{attribute 'linkalways'} 
{attribute 'no_explicit_call' := 'This FB is a CLASS and must be accessed using methods or properties'}
{attribute 'enable_dynamic_creation'}
FUNCTION_BLOCK JsonDeserializer EXTENDS Disposable IMPLEMENTS I_JsonDeserializer
VAR
	jsonParser : JsonDomParser;
	root : SJsonValue;
	garbageCollector : DeserializerGarbageCollector;
	nullNode : JsonDeserializerNullNode(THIS^);
	rootNode : I_Deserializer := nullNode;
	eventEmitter : EventEmitter;
END_VAR

METHOD PUBLIC Clone : I_Deserializer
VAR
	pClone : POINTER TO JsonDeserializer;
	jsonSize : UDINT;
	pJsonString : POINTER TO STRING;
END_VAR
pClone := __NEW(JsonDeserializer);
Clone := pClone^;

jsonSize := jsonParser.GetDocumentLength();

IF jsonSize = 0 THEN
	// no further cloning to do. 
	RETURN;
END_IF

pJsonString := __NEW(BYTE, jsonSize);

IF jsonParser.CopyDocument(pJsonString^, jsonSize) = 0 THEN
	__DELETE(pJsonString);
	RETURN;
END_IF

pClone^.TryLoad(pJsonString^);
__DELETE(pJsonString);
END_METHOD

METHOD PROTECTED CreateDeserializer : I_Deserializer
VAR_INPUT
	DeserializerRoot : SJsonValue;
END_VAR
VAR 
	pNode : POINTER TO JsonDeserializerNode;
END_VAR
pNode := __NEW(JsonDeserializerNode(
	ParentJsonDeserializer := THIS^,
	ParentJsonDomParser := jsonParser, 
	NodeRoot := DeserializerRoot, 
	ParentGarbageCollector := garbageCollector, 
	ParentNullDeserializer := nullNode)
);

CreateDeserializer := pNode^;
END_METHOD

METHOD PRIVATE EmitChangedEvent
VAR
	pJsonDeserializerChangedEvent : POINTER TO JsonDeserializerChangedEvent;
END_VAR
pJsonDeserializerChangedEvent := __NEW(JsonDeserializerChangedEvent(Target := THIS^));
eventEmitter.Emit('OnChanged', pJsonDeserializerChangedEvent^);
pJsonDeserializerChangedEvent^.Dispose();
END_METHOD

METHOD PRIVATE EmitDisposedEvent
VAR
	pJsonDeserializerDisposedEvent : POINTER TO JsonDeserializerDisposedEvent;
END_VAR
pJsonDeserializerDisposedEvent := __NEW(JsonDeserializerDisposedEvent(Target := THIS^));
eventEmitter.Emit('OnDisposed', pJsonDeserializerDisposedEvent^);
pJsonDeserializerDisposedEvent^.Dispose();
END_METHOD

METHOD FB_exit : BOOL
VAR_INPUT
	bInCopyCode : BOOL; // if TRUE, the exit method is called for exiting an instance that is copied afterwards (online change).
END_VAR
IF bInCopyCode THEN
	RETURN;
END_IF

Reset();
EmitDisposedEvent();
END_METHOD

METHOD GetArray : I_Deserializer
VAR_INPUT
END_VAR
GetArray := rootNode.GetArray();
END_METHOD

METHOD GetArrayEnumerator : I_DeserializerArrayForwardEnumerator
VAR_INPUT
END_VAR
GetArrayEnumerator := rootNode.GetArrayEnumerator();
END_METHOD

METHOD GetElementByIndex : I_Deserializer
VAR_INPUT
	Index : UDINT;
END_VAR
GetElementByIndex := rootNode.GetElementByIndex(Index);
END_METHOD

METHOD GetKeyArray : I_Deserializer
VAR_INPUT
	Key : T_MAXSTRING;
END_VAR
GetKeyArray := rootNode.GetKeyArray(Key);
END_METHOD

METHOD GetKeyObject : I_Deserializer
VAR_INPUT
	Key : T_MAXSTRING;
END_VAR
GetKeyObject := rootNode.GetKeyObject(Key);
END_METHOD

METHOD GetObject : I_Deserializer
VAR_INPUT
END_VAR
GetObject := rootNode.GetObject();
END_METHOD

METHOD GetObjectEnumerator : I_DeserializerObjectForwardEnumerator
VAR_INPUT
END_VAR
GetObjectEnumerator := rootNode.GetObjectEnumerator();
END_METHOD

METHOD PUBLIC OffEvent
VAR_INPUT
	EventName : T_MaxString;
	EventHandler : I_EventHandler;
END_VAR
eventEmitter.OffEvent(EventName, EventHandler);
END_METHOD

METHOD PUBLIC OnceEvent
VAR_INPUT
	EventName : T_MaxString;
	EventHandler : I_EventHandler;
END_VAR
eventEmitter.OnceEvent(EventName, EventHandler);
END_METHOD

METHOD PUBLIC OnEvent
VAR_INPUT
	EventName : T_MaxString;
	EventHandler : I_EventHandler;
END_VAR
eventEmitter.OnEvent(EventName, EventHandler);
END_METHOD

METHOD PUBLIC Reset
VAR_INPUT
END_VAR
jsonParser.NewDocument();
garbageCollector.Execute();
root := 0;
rootNode := nullNode;
EmitChangedEvent();
END_METHOD

METHOD TryDeserializeKeyToObject : BOOL
VAR_INPUT
	Key : T_MAXSTRING;
	Object : I_Deserializable;
	Feedback : I_DeserializerFeedback;
END_VAR
TryDeserializeKeyToObject := rootNode.TryDeserializeKeyToObject(Key,Object, Feedback);
END_METHOD

METHOD TryDeserializeToObject : BOOL
VAR_INPUT
	Object : I_Deserializable;
	Feedback : I_DeserializerFeedback;
END_VAR
TryDeserializeToObject := rootNode.TryDeserializeToObject(Object, Feedback);
END_METHOD

METHOD TryGetBase64 : BOOL
VAR_INPUT
	pBytes : POINTER TO BYTE;
	nBytes : DINT;
	Feedback : I_DeserializerFeedback;
END_VAR
TryGetBase64 := rootNode.TryGetBase64(pBytes, nBytes, Feedback);
END_METHOD

METHOD TryGetBool : BOOL
VAR_INPUT
	Destination : REFERENCE TO BOOL;
	Feedback : I_DeserializerFeedback;
END_VAR
TryGetBool := rootNode.TryGetBool(Destination, Feedback);
END_METHOD

METHOD TryGetByte : BOOL
VAR_INPUT
	Destination : REFERENCE TO BYTE;
	Feedback : I_DeserializerFeedback;
END_VAR
TryGetByte := rootNode.TryGetByte(Destination, Feedback);
END_METHOD

METHOD TryGetDateTime : BOOL
VAR_INPUT
	Destination : REFERENCE TO DATE_AND_TIME;
	Feedback : I_DeserializerFeedback;
END_VAR
TryGetDateTime := rootNode.TryGetDateTime(Destination, Feedback);
END_METHOD

METHOD TryGetDcTime : BOOL
VAR_INPUT
	Destination : REFERENCE TO DCTIME;
	Feedback : I_DeserializerFeedback;
END_VAR
TryGetDcTime := rootNode.TryGetDcTime(Destination, Feedback);
END_METHOD

METHOD TryGetDint : BOOL
VAR_INPUT
	Destination : REFERENCE TO DINT;
	Feedback : I_DeserializerFeedback;
END_VAR
TryGetDint := rootNode.TryGetDint(Destination, Feedback);
END_METHOD

METHOD TryGetDword : BOOL
VAR_INPUT
	Destination : REFERENCE TO DWORD;
	Feedback : I_DeserializerFeedback;
END_VAR
TryGetDword := rootNode.TryGetDword(Destination, Feedback);
END_METHOD

METHOD TryGetElementByIndex : BOOL
VAR_INPUT
	Index : UDINT;
	Destination : REFERENCE TO I_Deserializer;
	Feedback : I_DeserializerFeedback;
END_VAR
TryGetElementByIndex := rootNode.TryGetElementByIndex(Index, Destination, Feedback);
END_METHOD

METHOD TryGetFileTime : BOOL
VAR_INPUT
	Destination : REFERENCE TO FILETIME;
	Feedback : I_DeserializerFeedback;
END_VAR
TryGetFileTime := rootNode.TryGetFileTime(Destination, Feedback);
END_METHOD

METHOD TryGetHexAsBytes : BOOL
VAR_INPUT
	pBytes : POINTER TO BYTE;
	nBytes : DINT;
	Feedback : I_DeserializerFeedback;
END_VAR
TryGetHexAsBytes := rootNode.TryGetHexAsBytes(pBytes, nBytes, Feedback);
END_METHOD

METHOD TryGetInt : BOOL
VAR_INPUT
	Destination : REFERENCE TO INT;
	Feedback : I_DeserializerFeedback;
END_VAR
TryGetInt := rootNode.TryGetInt(Destination, Feedback);
END_METHOD

METHOD TryGetKeyBase64 : BOOL
VAR_INPUT
	Key : T_MAXSTRING;
	pBytes : POINTER TO BYTE;
	nBytes : DINT;
	Feedback : I_DeserializerFeedback;
END_VAR
TryGetKeyBase64 := rootNode.TryGetKeyBase64(Key, pBytes, nBytes, Feedback);
END_METHOD

METHOD TryGetKeyBool : BOOL
VAR_INPUT
	Key : T_MAXSTRING;
	Destination : REFERENCE TO BOOL;
	Feedback : I_DeserializerFeedback;
END_VAR
TryGetKeyBool := rootNode.TryGetKeyBool(Key, Destination, Feedback);
END_METHOD

METHOD TryGetKeyByte : BOOL
VAR_INPUT
	Key : T_MAXSTRING;
	Destination : REFERENCE TO BYTE;
	Feedback : I_DeserializerFeedback;
END_VAR
TryGetKeyByte := rootNode.TryGetKeyByte(Key, Destination, Feedback);
END_METHOD

METHOD TryGetKeyDateTime : BOOL
VAR_INPUT
	Key : T_MAXSTRING;
	Destination : REFERENCE TO DATE_AND_TIME;
	Feedback : I_DeserializerFeedback;
END_VAR
TryGetKeyDateTime := rootNode.TryGetKeyDateTime(Key, Destination, Feedback);
END_METHOD

METHOD TryGetKeyDcTime : BOOL
VAR_INPUT
	Key : T_MAXSTRING;
	Destination : REFERENCE TO DCTIME;
	Feedback : I_DeserializerFeedback;
END_VAR
TryGetKeyDcTime := rootNode.TryGetKeyDcTime(Key, Destination, Feedback);
END_METHOD

METHOD TryGetKeyDint : BOOL
VAR_INPUT
	Key : T_MAXSTRING;
	Destination : REFERENCE TO DINT;
	Feedback : I_DeserializerFeedback;
END_VAR
TryGetKeyDint := rootNode.TryGetKeyDint(Key, Destination, Feedback);
END_METHOD

METHOD TryGetKeyDword : BOOL
VAR_INPUT
	Key : T_MAXSTRING;
	Destination : REFERENCE TO DWORD;
	Feedback : I_DeserializerFeedback;
END_VAR
TryGetKeyDword := rootNode.TryGetKeyDword(Key, Destination, Feedback);
END_METHOD

METHOD TryGetKeyFileTime : BOOL
VAR_INPUT
	Key : T_MAXSTRING;
	Destination : REFERENCE TO FILETIME;
	Feedback : I_DeserializerFeedback;
END_VAR
TryGetKeyFileTime := rootNode.TryGetKeyFileTime(Key, Destination, Feedback);
END_METHOD

METHOD TryGetKeyHexAsBytes : BOOL
VAR_INPUT
	Key : T_MAXSTRING;
	pBytes : POINTER TO BYTE;
	nBytes : DINT;
	Feedback : I_DeserializerFeedback;
END_VAR
TryGetKeyHexAsBytes := rootNode.TryGetKeyHexAsBytes(Key, pBytes, nBytes, Feedback);
END_METHOD

METHOD TryGetKeyInt : BOOL
VAR_INPUT
	Key : T_MAXSTRING;
	Destination : REFERENCE TO INT;
	Feedback : I_DeserializerFeedback;
END_VAR
TryGetKeyInt := rootNode.TryGetKeyInt(Key, Destination, Feedback);
END_METHOD

METHOD TryGetKeyLint : BOOL
VAR_INPUT
	Key : T_MAXSTRING;
	Destination : REFERENCE TO LINT;
	Feedback : I_DeserializerFeedback;
END_VAR
TryGetKeyLint := rootNode.TryGetKeyLint(Key, Destination, Feedback);
END_METHOD

METHOD TryGetKeyLreal : BOOL
VAR_INPUT
	Key : T_MAXSTRING;
	Destination : REFERENCE TO LREAL;
	Feedback : I_DeserializerFeedback;
END_VAR
TryGetKeyLreal := rootNode.TryGetKeyLreal(Key, Destination, Feedback);
END_METHOD

METHOD TryGetKeyLtime : BOOL
VAR_INPUT
	Key : T_MAXSTRING;
	Destination : REFERENCE TO LTIME;
	Feedback : I_DeserializerFeedback;
END_VAR
TryGetKeyLtime := rootNode.TryGetKeyLtime(Key, Destination, Feedback);
END_METHOD

METHOD TryGetKeyLword : BOOL
VAR_INPUT
	Key : T_MAXSTRING;
	Destination : REFERENCE TO LWORD;
	Feedback : I_DeserializerFeedback;
END_VAR
TryGetKeyLword := rootNode.TryGetKeyLword(Key, Destination, Feedback);
END_METHOD

METHOD TryGetKeyReal : BOOL
VAR_INPUT
	Key : T_MAXSTRING;
	Destination : REFERENCE TO REAL;
	Feedback : I_DeserializerFeedback;
END_VAR
TryGetKeyReal := rootNode.TryGetKeyReal(Key, Destination, Feedback);
END_METHOD

METHOD TryGetKeySint : BOOL
VAR_INPUT
	Key : T_MAXSTRING;
	Destination : REFERENCE TO SINT;
	Feedback : I_DeserializerFeedback;
END_VAR
TryGetKeySint := rootNode.TryGetKeySint(Key, Destination, Feedback);
END_METHOD

METHOD TryGetKeyString : BOOL
VAR_INPUT
	Key : T_MAXSTRING;
	Destination : REFERENCE TO STRING;
	Feedback : I_DeserializerFeedback;
END_VAR
TryGetKeyString := rootNode.TryGetKeyString(Key, Destination, Feedback);
END_METHOD

METHOD TryGetKeyTime : BOOL
VAR_INPUT
	Key : T_MAXSTRING;
	Destination : REFERENCE TO TIME;
	Feedback : I_DeserializerFeedback;
END_VAR
TryGetKeyTime := rootNode.TryGetKeyTime(Key, Destination, Feedback);
END_METHOD

METHOD TryGetKeyTod : BOOL
VAR_INPUT
	Key : T_MAXSTRING;
	Destination : REFERENCE TO TOD;
	Feedback : I_DeserializerFeedback;
END_VAR
TryGetKeyTod := rootNode.TryGetKeyTod(Key, Destination, Feedback);
END_METHOD

METHOD TryGetKeyUdint : BOOL
VAR_INPUT
	Key : T_MAXSTRING;
	Destination : REFERENCE TO UDINT;
	Feedback : I_DeserializerFeedback;
END_VAR
TryGetKeyUdint := rootNode.TryGetKeyUdint(Key, Destination, Feedback);
END_METHOD

METHOD TryGetKeyUint : BOOL
VAR_INPUT
	Key : T_MAXSTRING;
	Destination : REFERENCE TO UINT;
	Feedback : I_DeserializerFeedback;
END_VAR
TryGetKeyUint := rootNode.TryGetKeyUint(Key, Destination, Feedback);
END_METHOD

METHOD TryGetKeyUlint : BOOL
VAR_INPUT
	Key : T_MAXSTRING;
	Destination : REFERENCE TO ULINT;
	Feedback : I_DeserializerFeedback;
END_VAR
TryGetKeyUlint := rootNode.TryGetKeyUlint(Key, Destination, Feedback);
END_METHOD

METHOD TryGetKeyUsint : BOOL
VAR_INPUT
	Key : T_MAXSTRING;
	Destination : REFERENCE TO USINT;
	Feedback : I_DeserializerFeedback;
END_VAR
TryGetKeyUsint := rootNode.TryGetKeyUsint(Key, Destination, Feedback);
END_METHOD

METHOD TryGetKeyWord : BOOL
VAR_INPUT
	Key : T_MAXSTRING;
	Destination : REFERENCE TO WORD;
	Feedback : I_DeserializerFeedback;
END_VAR
TryGetKeyWord := rootNode.TryGetKeyWord(Key, Destination, Feedback);
END_METHOD

METHOD TryGetLint : BOOL
VAR_INPUT
	Destination : REFERENCE TO LINT;
	Feedback : I_DeserializerFeedback;
END_VAR
TryGetLint := rootNode.TryGetLint(Destination, Feedback);
END_METHOD

METHOD TryGetLreal : BOOL
VAR_INPUT
	Destination : REFERENCE TO LREAL;
	Feedback : I_DeserializerFeedback;
END_VAR
TryGetLreal := rootNode.TryGetLreal(Destination, Feedback);
END_METHOD

METHOD TryGetLtime : BOOL
VAR_INPUT
	Destination : REFERENCE TO LTIME;
	Feedback : I_DeserializerFeedback;
END_VAR
TryGetLtime := rootNode.TryGetLtime(Destination, Feedback);
END_METHOD

METHOD TryGetLword : BOOL
VAR_INPUT
	Destination : REFERENCE TO LWORD;
	Feedback : I_DeserializerFeedback;
END_VAR
TryGetLword := rootNode.TryGetLword(Destination, Feedback);
END_METHOD

METHOD TryGetReal : BOOL
VAR_INPUT
	Destination : REFERENCE TO REAL;
	Feedback : I_DeserializerFeedback;
END_VAR
TryGetReal := rootNode.TryGetReal(Destination, Feedback);
END_METHOD

METHOD TryGetSint : BOOL
VAR_INPUT
	Destination : REFERENCE TO SINT;
	Feedback : I_DeserializerFeedback;
END_VAR
TryGetSint := rootNode.TryGetSint(Destination, Feedback);
END_METHOD

METHOD TryGetString : BOOL
VAR_INPUT
	Destination : REFERENCE TO STRING;
	Feedback : I_DeserializerFeedback;
END_VAR
TryGetString := rootNode.TryGetString(Destination, Feedback);
END_METHOD

METHOD TryGetTime : BOOL
VAR_INPUT
	Destination : REFERENCE TO TIME;
	Feedback : I_DeserializerFeedback;
END_VAR
TryGetTime := rootNode.TryGetTime(Destination, Feedback);
END_METHOD

METHOD TryGetTod : BOOL
VAR_INPUT
	Destination : REFERENCE TO TOD;
	Feedback : I_DeserializerFeedback;
END_VAR
TryGetTod := rootNode.TryGetTod(Destination, Feedback);
END_METHOD

METHOD TryGetUdint : BOOL
VAR_INPUT
	Destination : REFERENCE TO UDINT;
	Feedback : I_DeserializerFeedback;
END_VAR
TryGetUdint := rootNode.TryGetUdint(Destination, Feedback);
END_METHOD

METHOD TryGetUint : BOOL
VAR_INPUT
	Destination : REFERENCE TO UINT;
	Feedback : I_DeserializerFeedback;
END_VAR
TryGetUint := rootNode.TryGetUint(Destination, Feedback);
END_METHOD

METHOD TryGetUlint : BOOL
VAR_INPUT
	Destination : REFERENCE TO ULINT;
	Feedback : I_DeserializerFeedback;
END_VAR
TryGetUlint := rootNode.TryGetUlint(Destination, Feedback);
END_METHOD

METHOD TryGetUsint : BOOL
VAR_INPUT
	Destination : REFERENCE TO USINT;
	Feedback : I_DeserializerFeedback;
END_VAR
TryGetUsint := rootNode.TryGetUsint(Destination, Feedback);
END_METHOD

METHOD TryGetWord : BOOL
VAR_INPUT
	Destination : REFERENCE TO WORD;
	Feedback : I_DeserializerFeedback;
END_VAR
TryGetWord := rootNode.TryGetWord(Destination, Feedback);
END_METHOD

METHOD PUBLIC TryLoad : BOOL
VAR_INPUT
	SerializedData : REFERENCE TO STRING;;
END_VAR
Reset();
EmitChangedEvent();

root := jsonParser.ParseDocument(SerializedData);
IF root = 0 THEN
	RETURN;
END_IF

rootNode := CreateDeserializer(root);
TryLoad := TRUE;
END_METHOD

END_FUNCTION_BLOCK

(* stored: Version 1.1.0.1, ProductVersion 3.1.4024.13
   POU JsonDeserializer: Id {33607e16-d857-42ff-a777-ee399a72a022}, SpecialFunc None
   Folder Destructor: Id {25e81e5b-1097-4887-b433-bd17750805b6}
   Folder Protected: Id {9baf6261-9616-4d4e-919a-e38cd3fecd6b}
   Method Clone: Id {6af19bf6-271b-48fa-bfd5-c84e2e38f2ff}
   Method CreateDeserializer: Id {f47db19e-f95c-4af5-aa9e-767fe9d54a57}
   Method EmitChangedEvent: Id {a8f8ce98-9a65-4156-b899-af3c07a7184f}
   Method EmitDisposedEvent: Id {4fa93604-636c-45c6-b1ff-952cb2890027}
   Method FB_exit: Id {4398bb00-38b7-4fe4-aa40-d948cb60b2a6}
   Method GetArray: Id {32df193d-6d43-4275-ab94-3dc2b51c2046}
   Method GetArrayEnumerator: Id {b301d3aa-0537-45d8-8a0d-bc196dc5c2e1}
   Method GetElementByIndex: Id {3791a964-baca-4d3d-9968-3575b0604fce}
   Method GetKeyArray: Id {fe8706d8-759e-4a7f-9edf-ce884f0686b1}
   Method GetKeyObject: Id {957a487d-4d6e-4520-bf02-4254a13a84e2}
   Method GetObject: Id {dbad7a18-a1a1-4eb3-a1b7-ca71e2e9833a}
   Method GetObjectEnumerator: Id {d4ef2b7e-99de-4b5b-9025-9dc1826653e5}
   Method OffEvent: Id {0f81a8a8-ffaa-42c0-ad6e-9ad5d9928de4}
   Method OnceEvent: Id {582317cd-b61d-4471-8f87-6f33eebfd143}
   Method OnEvent: Id {e06b2f22-0254-4153-982f-2ed6270cb287}
   Method Reset: Id {652b36eb-59e6-415a-8da0-4e52da0b1670}
   Method TryDeserializeKeyToObject: Id {f8874143-c444-4dba-8b46-312d2aacbb62}
   Method TryDeserializeToObject: Id {d051848e-a1a9-4787-82f4-96ef3b35c8c9}
   Method TryGetBase64: Id {6443636e-51b0-46c1-b03f-c4cd6ba1dbf3}
   Method TryGetBool: Id {f4ac3f58-ce4d-4413-b0ba-726a0a7897b6}
   Method TryGetByte: Id {e53c8f9e-dcd5-444e-a88e-1ab8419aebc3}
   Method TryGetDateTime: Id {9485f7fb-5cb3-425d-81a1-095442dc10f4}
   Method TryGetDcTime: Id {184628de-186e-4167-9b8d-cb860b321fb4}
   Method TryGetDint: Id {e8bb9f39-5f29-49ed-be41-bf9f49e5300b}
   Method TryGetDword: Id {08f30628-1d86-43ea-96ad-5cb92af283b7}
   Method TryGetElementByIndex: Id {474769dc-4905-0ab2-0cc8-226e8072f161}
   Method TryGetFileTime: Id {f5f266cd-a2bf-44cb-bc66-3de5433dcfa9}
   Method TryGetHexAsBytes: Id {cd1860a0-455c-4ea0-845b-a011925107f9}
   Method TryGetInt: Id {b5b52ba4-6535-4abf-8491-6e5079e5f5e7}
   Method TryGetKeyBase64: Id {78834054-7389-4b1b-a140-72e318e8511c}
   Method TryGetKeyBool: Id {c54c4743-d9f1-4600-8cd1-8f68b966bbb4}
   Method TryGetKeyByte: Id {8629d883-dc72-472a-808f-9a9bb185fb5e}
   Method TryGetKeyDateTime: Id {5841be57-1eb3-4723-ad01-22740f06a693}
   Method TryGetKeyDcTime: Id {a2484634-7ec7-430e-909a-54084f7ac095}
   Method TryGetKeyDint: Id {1897ce6f-a6f7-40df-ae1c-0ab8575a4cf9}
   Method TryGetKeyDword: Id {c02fef7c-d08f-4f2f-9fc5-12612b88cbff}
   Method TryGetKeyFileTime: Id {5470f571-9ab2-419f-aac3-5ec7fa739940}
   Method TryGetKeyHexAsBytes: Id {f7505922-db31-4e54-abc9-a76cc91bac25}
   Method TryGetKeyInt: Id {0712ded5-f2f8-4793-9ae8-098609af9f3e}
   Method TryGetKeyLint: Id {4b43a83a-674c-48c8-a661-dc009a0dde7e}
   Method TryGetKeyLreal: Id {08a9d73c-43ea-447e-86b2-f4abcdce24af}
   Method TryGetKeyLtime: Id {6a80c1d1-8d7e-46ba-81ca-af1ea8a9ee02}
   Method TryGetKeyLword: Id {ff81c406-b573-41a1-a4b6-c7153d028ddf}
   Method TryGetKeyReal: Id {20f6bb54-fd66-4d4f-8187-84b31223cd71}
   Method TryGetKeySint: Id {064b3089-80fa-44d6-8f6d-59cc727ea997}
   Method TryGetKeyString: Id {8e34a995-537d-4c0c-b13f-bd424b3e589a}
   Method TryGetKeyTime: Id {36761ef9-1461-449a-a02c-08088b4b7b03}
   Method TryGetKeyTod: Id {278af3a0-ffa2-45b7-a712-3c9febfa2f66}
   Method TryGetKeyUdint: Id {a51b96a5-1e14-42eb-8289-6961e8165ba4}
   Method TryGetKeyUint: Id {2af7b8ba-3b38-43b5-9cef-e203cac32bce}
   Method TryGetKeyUlint: Id {d3f4de97-f59c-4512-a9a0-6e2999c24f43}
   Method TryGetKeyUsint: Id {af9c46be-c08d-47d7-a792-5013a98e8bbb}
   Method TryGetKeyWord: Id {e4908f50-c709-4d4b-a9e4-b014057d9704}
   Method TryGetLint: Id {ef192691-d277-4a5a-9ff0-5e661d0f3753}
   Method TryGetLreal: Id {e15238c8-65c7-40c2-a47a-4343df0dbfba}
   Method TryGetLtime: Id {75bdc86c-ba76-4c13-80a7-7c69b1f5fd2f}
   Method TryGetLword: Id {98ff927b-c265-42c4-a02a-ae6164a28065}
   Method TryGetReal: Id {f658ad1c-ccf1-4da6-99f1-dd9c659afd24}
   Method TryGetSint: Id {722f5830-4351-4acd-a3b4-024f05358d74}
   Method TryGetString: Id {de4e33a0-ab56-4d57-ad2a-2035c735b78c}
   Method TryGetTime: Id {1ab23048-c202-493d-b3ae-ba72573f1eb2}
   Method TryGetTod: Id {046e14a6-cd7f-4165-b5cb-7de9f6dae441}
   Method TryGetUdint: Id {ef71d1b1-0835-497d-8e60-af9216234170}
   Method TryGetUint: Id {0d4f5b05-60af-45e2-8771-535598c24115}
   Method TryGetUlint: Id {a52011fc-a47c-4f90-bb7d-f7807961f22e}
   Method TryGetUsint: Id {8d7ab32d-181a-425c-9e2b-9fc4f8e29626}
   Method TryGetWord: Id {a3892e80-ad23-4c26-b8d0-b4d8f71a2c85}
   Method TryLoad: Id {6a1f9be2-30a8-476b-9f1e-f75bb911b849} *)
